// SIMATIC S7-200 SMART project (STEP 7-Micro/WIN SMART), CPU SR20

SYMBOL_TABLE 表格 1
点火命令1            M0.0
点火成功信号1          M0.1
故障复位1            M0.2     // 输出
点火变压器1           M1.0     // 输出
点火电磁阀1           M1.1     // 输出
报警1              M1.2     // 输出
END_SYMBOL_TABLE

SYMBOL_TABLE 系统符号
Always_On        SM0.0    // 始终接通
END_SYMBOL_TABLE

ORGANIZATION_BLOCK MAIN:OB1
TITLE=程序注释
BEGIN
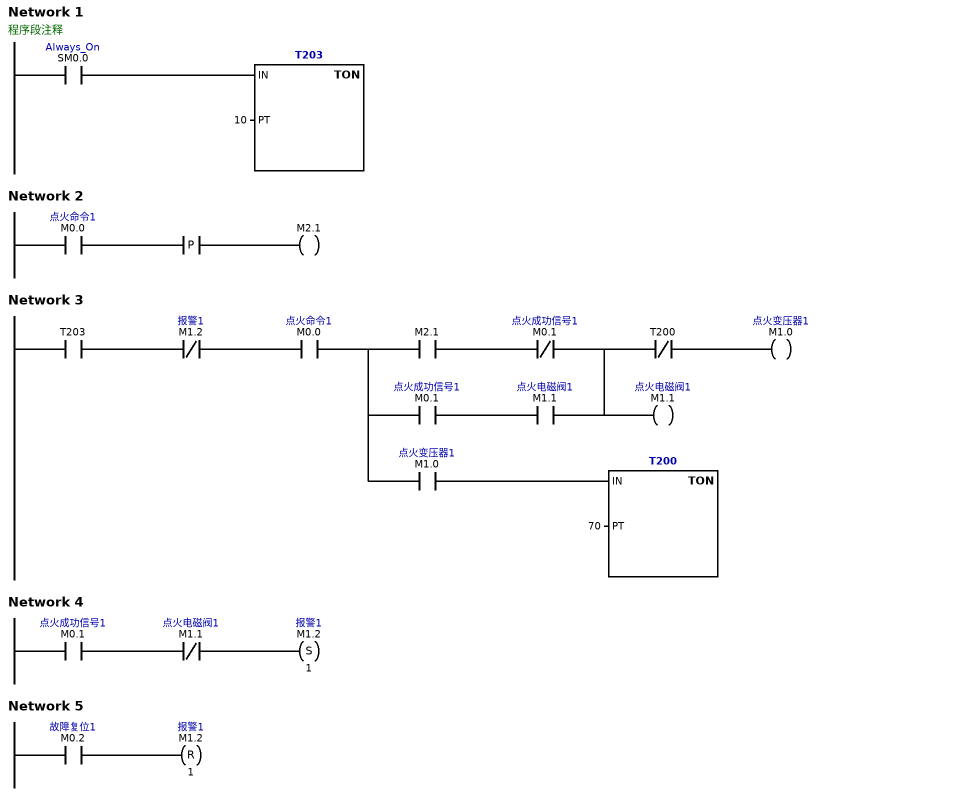
Network 1
// 程序段注释
LD     Always_On:SM0.0
TON    T203, 10
Network 2
LD     点火命令1:M0.0
EU
=      M2.1
Network 3
// (network saved uncompiled; LAD cells follow)
// row 0: c0 -| |- T203  c1 -|/|- 报警1:M1.2  c2 -| |- 点火命令1:M0.0 v  c3 -| |- M2.1  c4 -|/|- 点火成功信号1:M0.1 v  c5 -|/|- T200  c6 -( ) 点火变压器1:M1.0
// row 1: c2 ^v  c3 -| |- 点火成功信号1:M0.1  c4 -| |- 点火电磁阀1:M1.1 ^  c5 -( ) 点火电磁阀1:M1.1
// row 2: c2 ^  c3 -| |- 点火变压器1:M1.0  c4 --  c5 [TON T200 IN:=power@row2, PT:=70]
// row 3: c5 [box]
Network 4
LD     点火成功信号1:M0.1
AN     点火电磁阀1:M1.1
S      报警1:M1.2, 1
Network 5
// (network saved uncompiled; LAD cells follow)
// row 0: c0 -| |- 故障复位1:M0.2  c1 -(R) 报警1:M1.2, 1
END_ORGANIZATION_BLOCK
